// TIA Portal V19 export
DATA_BLOCK "G120 Comm_DB"   // DB17
// stored: InstanceOfName G120 Comm, InstanceOfType FB
"G120 Comm"
   // VAR_OUTPUT
   //    AnalogInput : Real;
   // END_VAR
   // VAR
   //    WRREC_Instance { S7_SetPoint := 'True'} : WRREC;
   //    RDREC_Instance { S7_SetPoint := 'True'} : RDREC;
   //    WriteRecord : Struct
   //       Static_1 { S7_SetPoint := 'True'} : "HEADER";
   //       Static_2 { S7_SetPoint := 'True'} : "PARAMETERADDR";
   //    END_STRUCT;
   //    ReadRecord : Struct
   //       data : Array[0..5] of Byte;
   //       Value : Real;
   //    END_STRUCT;
   // END_VAR
BEGIN
END_DATA_BLOCK
